# EPICS substitutions: MERCURY_ITC/MERCURY-IOC-01App/Db/main_unit.substitutions
file $(MERCURY_ITC)/db/MercuryiTC-SCPI.template
{
pattern {P, Q, PORT}
	{\$(P):MERCURY, 01, \$(PORT)}
}
